// TIA Portal V18 export
VAR_GLOBAL   // PLC tag table "Default tag table"
   Tag_1 AT %I0.1 : Bool;
END_VAR
